FUNCTION_BLOCK PR_02 (* Insert Product Type *)
  (* Standard: 61499-2 *)
  (* Version 1.0, 2022-12-15, AK124017 *)
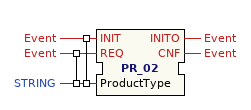
  EVENT_INPUT
    INIT WITH ProductType; (* Initialization Request *)
    REQ WITH ProductType; (* Normal Execution Request *)
  END_EVENT
  EVENT_OUTPUT
    INITO; (* Initialization Confirm *)
    CNF; (* Execution Confirmation *)
  END_EVENT
  VAR_INPUT
    ProductType : STRING; (* Type of Product *)
  END_VAR
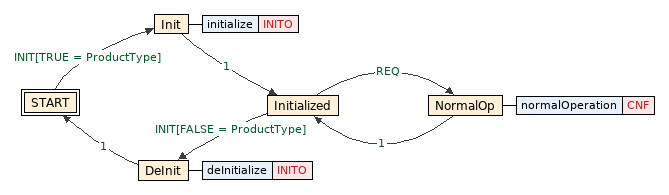
  EC_STATES
    START; (* Initial State *)
    Init : initialize -> INITO; (* Initialization *)
    NormalOp : normalOperation -> CNF; (* Normal execution *)
    Initialized;
    DeInit : deInitialize -> INITO;
  END_STATES
  EC_TRANSITIONS
    START TO Init := INIT[TRUE = ProductType];
    Init TO Initialized := 1;
    Initialized TO NormalOp := REQ;
    NormalOp TO Initialized := 1;
    DeInit TO START := 1;
    Initialized TO DeInit := INIT[FALSE = ProductType];
  END_TRANSITIONS
  ALGORITHM initialize IN ST:

  END_ALGORITHM
  ALGORITHM deInitialize IN ST:

  END_ALGORITHM
  ALGORITHM normalOperation IN ST:

  END_ALGORITHM
END_FUNCTION_BLOCK
